FUNCTION GetMaterialLength : LREAL
VAR_INPUT
	material : STRING;
END_VAR
VAR
	i : INT;
END_VAR

FOR i:=0 TO CONSTS.numMaterials BY 1 DO
	IF CONSTS.allMaterials[i].code = material THEN
		getMaterialLength := CONSTS.allMaterials[i].length;
		RETURN;
	END_IF
END_FOR
//otherwise, return 0
GetMaterialLength := 0;

END_FUNCTION

(* stored: Version 1.1.0.1, ProductVersion 3.1.4024.11
   POU GetMaterialLength: Id {3168ca70-88ff-44da-a8e2-6eae63f5c2da}, SpecialFunc None *)
